// TIA Portal V20 export
// export: Created 2025-12-01T14:56:48.0251132Z, ExportSetting None, DisplayName Totally Integrated Automation Portal, DisplayVersion V20 Update 3, DisplayName TIA Portal Openness, DisplayVersion V20 Update 3, DisplayName TIA Portal Version Control Interface, DisplayVersion V20 Update 3, DisplayName STEP 7 Professional, DisplayVersion V20 Update 3, DisplayName STEP 7 Safety, DisplayVersion V20 Update 2, DisplayName WinCC Basic/Comfort/Advanced, DisplayVersion V20 Update 3, DisplayName WinCC Professional, DisplayVersion V20 Update 3, DisplayName WinCC Unified, DisplayVersion V20 Update 3
FUNCTION_BLOCK "FB101_GIRO_Mesa"   // FB101, LAD
TITLE = FB101
{ S7_Optimized_Access := 'FALSE' }
// FB complementaria a cualquier FB de mesa, solo gestiona el giro.
// stored: AutoNumber false, SetENOAutomatically false
   VAR_INPUT
      Mesa : UInt;   // Mesa de la FB
      Error_Tx : Bool;   // Error en el Tx
      EnTension : Bool;   // Existe Tension en la Mesa
      FalloVar_MG : Bool;   // Señal VAR ok
      MG_EnMovimiento : Bool;   // Señal VAR giro en curso
      PosMG_0 : Bool;   // Detector Posicion 0
      PosMG_90 : Bool;   // Detector Posicion 90
      PosMG_180 : Bool;   // Detector Posicion 180
      PosMG_270 : Bool;   // Detector Posicion 270
      pHsPR : Bool;   // pHs de Protrusion de la Mesa. Nota: No existe >> ON
      Movhabi0_90 : Bool;   // Habilitar zona movimiento entre 0 y 90º
      Movhabi90_180 : Bool;   // Habilitar zona movimiento entre 90 y 180º
      Movhabi180_270 : Bool;   // Habilitar zona movimiento entre 180 y 270º
      Movhabi270_0 : Bool;   // Habilitar zona movimiento entre 270 y 0º
      Mx_VelocidadLenta_In : Bool;   // Forzar velocidad lenta
      OrdPos_0 : Bool;   // Orden ir a Posicion 0
      OrdPos_90 : Bool;   // Orden ir a Posicion 90
      OrdPos_180 : Bool;   // Orden ir a Posicion 180
      OrdPos_270 : Bool;   // Orden ir a Posicion 270
      V_TOut_MG_90º : Int := 15;   // Timeout para un movimiento de 90º
      V_TOut_MG_180º : Int := 30;   // Timeout para un movimiento de 180º
      V_TOut_MG_270º : Int := 45;   // Timeout para un movimiento de 270º
      V_TOut_MG_BusqPos : Int := 15;   // Timeout para busqueda de posición en velo lenta
      V_CNT_PerdidaPos : Int := 5000;   // Perdida de posición
      V_PasoLenta_Mov90 : Int := 800;   // Cambio de velocidad durante un movimiento de 90º
      V_PasoLenta_Mov180 : Int := 1800;   // Cambio de velocidad durante un movimiento de 180º
      V_PasoLenta_Mov270 : Int := 2800;   // Cambio de velocidad durante un movimiento de 270º
      V_CNTSeg_AusPos : Int := 3000;   // Contador de seguridade posicionamiento
   END_VAR
   VAR
      MGiro_EnPos0 : Bool;   // Mesa Giro en posición 0º
      MGiro_EnPos90 : Bool;   // Mesa Giro en posición 90º
      MGiro_EnPos180 : Bool;   // Mesa Giro en posición 180º
      MGiro_EnPos270 : Bool;   // Mesa Giro en posición 270º
      PosOK { ExternalVisible := 'False'} : Bool;
      Orden_AvGiro : Bool;   // Orden de Avance (sentido agujas reloj)
      Orden_RtGiro : Bool;   // Orden de Retroceso (sentido inverso agujas reloj)
      DestinoPos0 : Bool;   // Destino a la posición 0º
      DestinoPos90 : Bool;   // Destino a la posición 90º
      DestinoPos180 : Bool;   // Destino a la posición 180º
      DestinoPos270 : Bool;   // Destino a la posición 270º
      Giro90º : Bool;   // Distancia de giro en grados desde origen hasta destino
      Giro180º : Bool;   // Distancia de giro en grados desde origen hasta destino
      Giro270º : Bool;   // Distancia de giro en grados desde origen hasta destino
      Pos_Desconocida : Bool;
      Pos_Conocida : Bool;
      Destino_Desconocido : Bool;
      Busq_Posicion : Bool;
      Mem_Busq_Posicion : Bool;
      VelocidadLenta { ExternalAccessible := 'False'; ExternalVisible := 'False'; ExternalWritable := 'False'} : Bool;
      MA_Avance_MG : Bool;   // Avance = ir de 0º a 360º
      MA_Retroceso_MG : Bool;   // Retroceso = volver de 360º a 0
      VelocidadRapida_MG : Bool;
      CNT_Paso_Lenta : Int;
      CNTSeg_AusPos { S7_SetPoint := 'True'} : "FB910_CNT_UHS";
      TMP_EnTension { S7_SetPoint := 'True'} : "FB910_CNT_UHS";
      TOut_MG { S7_SetPoint := 'True'} : "FB910_CNT_UHS";
      TOut_MG_BusPos { S7_SetPoint := 'True'} : "FB910_CNT_UHS";
      CNT_PerdidaPos { S7_SetPoint := 'True'} : "FB910_CNT_UHS";
   END_VAR
   VAR_TEMP
      EstadoZona : "EstadoZona";   // Estado de Zona de la Mesa
      EstadoVI : "EstadosMesa";   // Estado del Vehiculo Inteliguente de la Mesa
      ConfigFB : "UDT_ConfigFB";   // Configuracion de la FB de la Mesa
      V_TOut_MG : Int;
      Basura : Bool;
   END_VAR
   VAR_TEMP   // added for the SCL form of the ladder/FBD networks
      _w1 : Bool;
   END_VAR
BEGIN

REGION Network 1: INICIALIZAR - Recoger las Variables de Estado de la Mesa
   // Se recoge - Estado_CBx
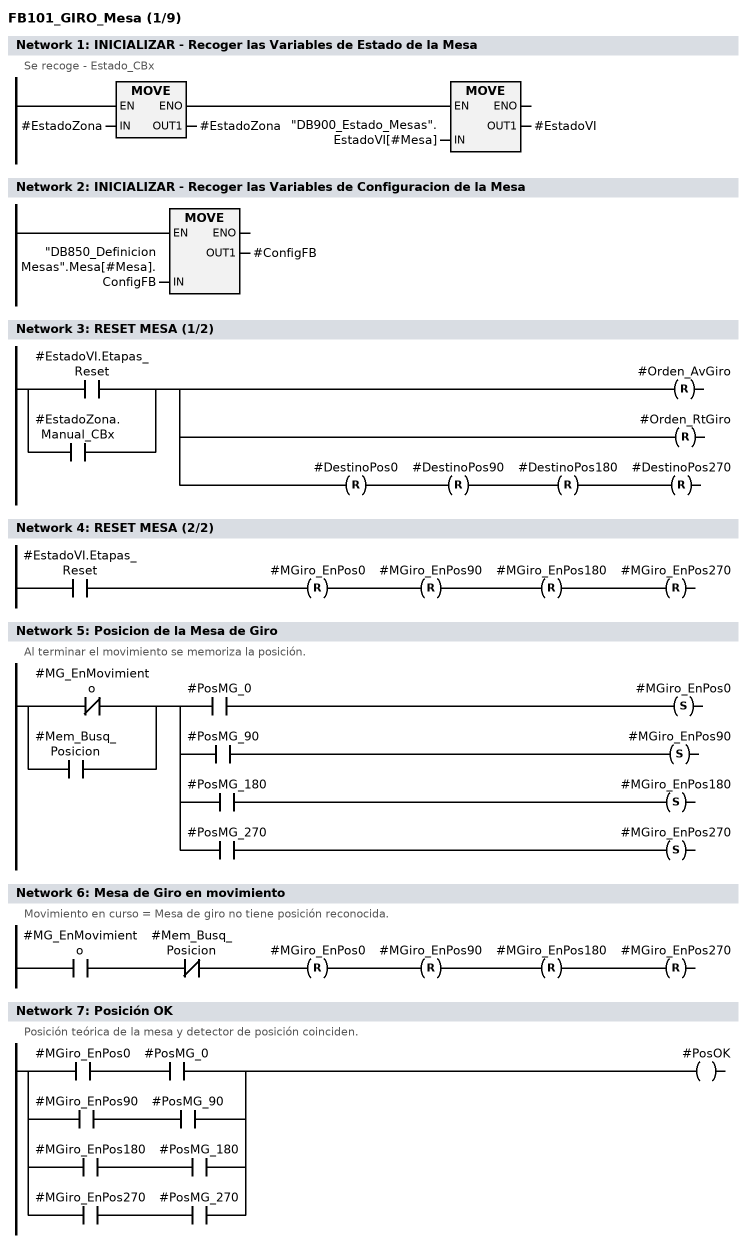
   RUNG wire#powerrail
      Move(in := #EstadoZona, out1 => #EstadoZona)
      Move(in := "DB900_Estado_Mesas".EstadoVI[#Mesa], out1 => #EstadoVI)
   END_RUNG
   // the same network as SCL:
   #EstadoZona := #EstadoZona;
   #EstadoVI := "DB900_Estado_Mesas".EstadoVI[#Mesa];
END_REGION

REGION Network 2: INICIALIZAR - Recoger las Variables de Configuracion de la Mesa
   RUNG wire#powerrail
      Move(in := "DB850_DefinicionMesas".Mesa[#Mesa].ConfigFB, out1 => #ConfigFB)
   END_RUNG
   // the same network as SCL:
   #ConfigFB := "DB850_DefinicionMesas".Mesa[#Mesa].ConfigFB;
END_REGION

REGION Network 3: RESET MESA (1/2)
   RUNG wire#powerrail
      Contact( #EstadoVI.Etapas_Reset )
      wire#w1
      R_Coil( #Orden_AvGiro )
   END_RUNG
   RUNG wire#powerrail
      Contact( #EstadoZona.Manual_CBx )
   END_RUNG wire#w1
   RUNG wire#w1
      R_Coil( #Orden_RtGiro )
   END_RUNG
   RUNG wire#w1
      R_Coil( #DestinoPos0 )
      R_Coil( #DestinoPos90 )
      R_Coil( #DestinoPos180 )
      R_Coil( #DestinoPos270 )
   END_RUNG
   // the same network as SCL:
   IF #EstadoVI.Etapas_Reset OR #EstadoZona.Manual_CBx THEN
       #Orden_AvGiro := FALSE;
       #Orden_RtGiro := FALSE;
       #DestinoPos0 := FALSE;
       #DestinoPos90 := FALSE;
       #DestinoPos180 := FALSE;
       #DestinoPos270 := FALSE;
   END_IF;
END_REGION

REGION Network 4: RESET MESA (2/2)
   RUNG wire#powerrail
      Contact( #EstadoVI.Etapas_Reset )
      R_Coil( #MGiro_EnPos0 )
      R_Coil( #MGiro_EnPos90 )
      R_Coil( #MGiro_EnPos180 )
      R_Coil( #MGiro_EnPos270 )
   END_RUNG
   // the same network as SCL:
   IF #EstadoVI.Etapas_Reset THEN
       #MGiro_EnPos0 := FALSE;
       #MGiro_EnPos90 := FALSE;
       #MGiro_EnPos180 := FALSE;
       #MGiro_EnPos270 := FALSE;
   END_IF;
END_REGION

REGION Network 5: Posicion de la Mesa de Giro
   // Al terminar el movimiento se memoriza la posición.
   RUNG wire#powerrail
      I_Contact( #MG_EnMovimiento )
      wire#w1
      Contact( #PosMG_0 )
      S_Coil( #MGiro_EnPos0 )
   END_RUNG
   RUNG wire#powerrail
      Contact( #Mem_Busq_Posicion )
   END_RUNG wire#w1
   RUNG wire#w1
      Contact( #PosMG_90 )
      S_Coil( #MGiro_EnPos90 )
   END_RUNG
   RUNG wire#w1
      Contact( #PosMG_180 )
      S_Coil( #MGiro_EnPos180 )
   END_RUNG
   RUNG wire#w1
      Contact( #PosMG_270 )
      S_Coil( #MGiro_EnPos270 )
   END_RUNG
   // the same network as SCL:
   #_w1 := NOT #MG_EnMovimiento OR #Mem_Busq_Posicion;
   IF #_w1 AND #PosMG_0 THEN #MGiro_EnPos0 := TRUE; END_IF;
   IF #_w1 AND #PosMG_90 THEN #MGiro_EnPos90 := TRUE; END_IF;
   IF #_w1 AND #PosMG_180 THEN #MGiro_EnPos180 := TRUE; END_IF;
   IF #_w1 AND #PosMG_270 THEN #MGiro_EnPos270 := TRUE; END_IF;
END_REGION

REGION Network 6: Mesa de Giro en movimiento
   // Movimiento en curso = Mesa de giro no tiene posición reconocida.
   RUNG wire#powerrail
      Contact( #MG_EnMovimiento )
      I_Contact( #Mem_Busq_Posicion )
      R_Coil( #MGiro_EnPos0 )
      R_Coil( #MGiro_EnPos90 )
      R_Coil( #MGiro_EnPos180 )
      R_Coil( #MGiro_EnPos270 )
   END_RUNG
   // the same network as SCL:
   IF #MG_EnMovimiento AND NOT #Mem_Busq_Posicion THEN
       #MGiro_EnPos0 := FALSE;
       #MGiro_EnPos90 := FALSE;
       #MGiro_EnPos180 := FALSE;
       #MGiro_EnPos270 := FALSE;
   END_IF;
END_REGION

REGION Network 7: Posición OK
   // Posición teórica de la mesa y detector de posición coinciden.
   RUNG wire#powerrail
      Contact( #MGiro_EnPos0 )
      Contact( #PosMG_0 )
      wire#w1
      Coil( #PosOK )
   END_RUNG
   RUNG wire#powerrail
      Contact( #MGiro_EnPos90 )
      Contact( #PosMG_90 )
   END_RUNG wire#w1
   RUNG wire#powerrail
      Contact( #MGiro_EnPos180 )
      Contact( #PosMG_180 )
   END_RUNG wire#w1
   RUNG wire#powerrail
      Contact( #MGiro_EnPos270 )
      Contact( #PosMG_270 )
   END_RUNG wire#w1
   // the same network as SCL:
   #PosOK := (#MGiro_EnPos0 AND #PosMG_0) OR (#MGiro_EnPos90 AND #PosMG_90) OR (#MGiro_EnPos180 AND #PosMG_180) OR (#MGiro_EnPos270 AND #PosMG_270);
END_REGION

REGION Network 8: Destino Desconocido // Posicion desconocida // Posicion Conocida
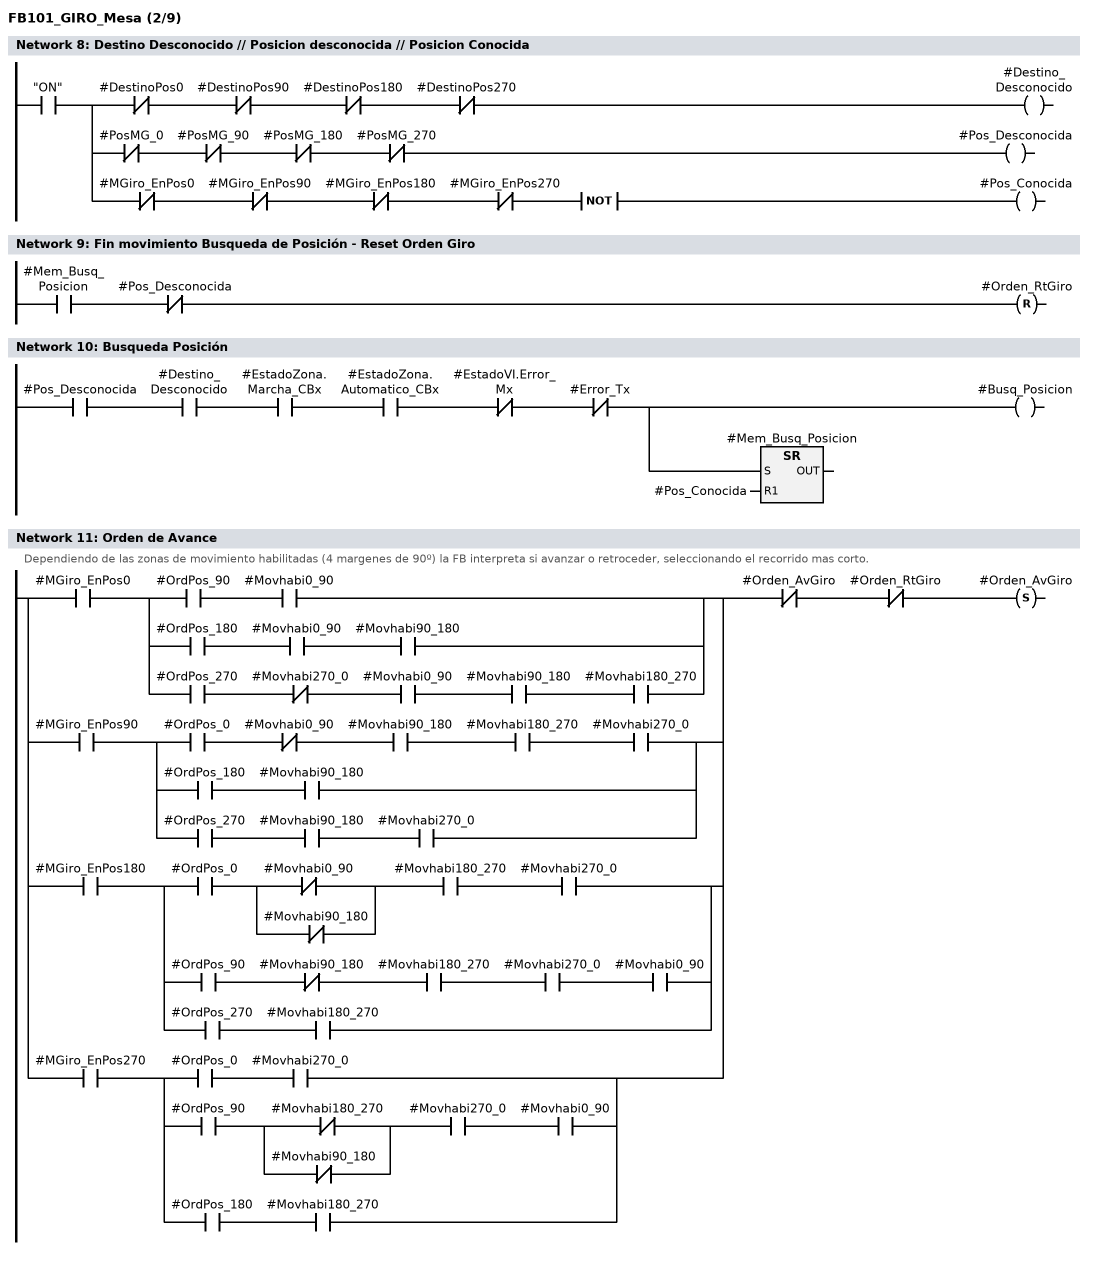
   RUNG wire#powerrail
      Contact( "ON" )
      wire#w1
      I_Contact( #DestinoPos0 )
      I_Contact( #DestinoPos90 )
      I_Contact( #DestinoPos180 )
      I_Contact( #DestinoPos270 )
      Coil( #Destino_Desconocido )
   END_RUNG
   RUNG wire#w1
      I_Contact( #PosMG_0 )
      I_Contact( #PosMG_90 )
      I_Contact( #PosMG_180 )
      I_Contact( #PosMG_270 )
      Coil( #Pos_Desconocida )
   END_RUNG
   RUNG wire#w1
      I_Contact( #MGiro_EnPos0 )
      I_Contact( #MGiro_EnPos90 )
      I_Contact( #MGiro_EnPos180 )
      I_Contact( #MGiro_EnPos270 )
      Not()
      Coil( #Pos_Conocida )
   END_RUNG
   // the same network as SCL:
   #Destino_Desconocido := "ON" AND NOT #DestinoPos0 AND NOT #DestinoPos90 AND NOT #DestinoPos180 AND NOT #DestinoPos270;
   #Pos_Desconocida := "ON" AND NOT #PosMG_0 AND NOT #PosMG_90 AND NOT #PosMG_180 AND NOT #PosMG_270;
   #Pos_Conocida := NOT ("ON" AND NOT #MGiro_EnPos0 AND NOT #MGiro_EnPos90 AND NOT #MGiro_EnPos180 AND NOT #MGiro_EnPos270);
END_REGION

REGION Network 9: Fin movimiento Busqueda de Posición - Reset Orden Giro
   RUNG wire#powerrail
      Contact( #Mem_Busq_Posicion )
      I_Contact( #Pos_Desconocida )
      R_Coil( #Orden_RtGiro )
   END_RUNG
   // the same network as SCL:
   IF #Mem_Busq_Posicion AND NOT #Pos_Desconocida THEN #Orden_RtGiro := FALSE; END_IF;
END_REGION

REGION Network 10: Busqueda Posición
   RUNG wire#powerrail
      Contact( #Pos_Desconocida )
      Contact( #Destino_Desconocido )
      Contact( #EstadoZona.Marcha_CBx )
      Contact( #EstadoZona.Automatico_CBx )
      I_Contact( #EstadoVI.Error_Mx )
      I_Contact( #Error_Tx )
      wire#w1
      Coil( #Busq_Posicion )
   END_RUNG
   RUNG wire#w1
      S_SR(operand := #Mem_Busq_Posicion, r1 := #Pos_Conocida)
   END_RUNG
   // the same network as SCL:
   #Busq_Posicion := #Pos_Desconocida AND #Destino_Desconocido AND #EstadoZona.Marcha_CBx AND #EstadoZona.Automatico_CBx AND NOT #EstadoVI.Error_Mx AND NOT #Error_Tx;
   IF #Busq_Posicion THEN
       #Mem_Busq_Posicion := TRUE;   // SR flip-flop
   END_IF;
   IF #Pos_Conocida THEN #Mem_Busq_Posicion := FALSE; END_IF;
END_REGION

REGION Network 11: Orden de Avance
   // Dependiendo de las zonas de movimiento habilitadas (4 margenes de 90º) la FB interpreta si avanzar o retroceder, seleccionando el recorrido mas corto.
   RUNG wire#powerrail
      Contact( #MGiro_EnPos0 )
      wire#w1
      Contact( #OrdPos_90 )
      Contact( #Movhabi0_90 )
      wire#w2
      I_Contact( #Orden_AvGiro )
      I_Contact( #Orden_RtGiro )
      S_Coil( #Orden_AvGiro )
   END_RUNG
   RUNG wire#w1
      Contact( #OrdPos_180 )
      Contact( #Movhabi0_90 )
      Contact( #Movhabi90_180 )
   END_RUNG wire#w2
   RUNG wire#w1
      Contact( #OrdPos_270 )
      I_Contact( #Movhabi270_0 )
      Contact( #Movhabi0_90 )
      Contact( #Movhabi90_180 )
      Contact( #Movhabi180_270 )
   END_RUNG wire#w2
   RUNG wire#powerrail
      Contact( #MGiro_EnPos90 )
      wire#w3
      Contact( #OrdPos_0 )
      I_Contact( #Movhabi0_90 )
      Contact( #Movhabi90_180 )
      Contact( #Movhabi180_270 )
      Contact( #Movhabi270_0 )
   END_RUNG wire#w2
   RUNG wire#w3
      Contact( #OrdPos_180 )
      Contact( #Movhabi90_180 )
   END_RUNG wire#w2
   RUNG wire#w3
      Contact( #OrdPos_270 )
      Contact( #Movhabi90_180 )
      Contact( #Movhabi270_0 )
   END_RUNG wire#w2
   RUNG wire#powerrail
      Contact( #MGiro_EnPos180 )
      wire#w4
      Contact( #OrdPos_0 )
      wire#w5
      I_Contact( #Movhabi0_90 )
      wire#w6
      Contact( #Movhabi180_270 )
      Contact( #Movhabi270_0 )
   END_RUNG wire#w2
   RUNG wire#w5
      I_Contact( #Movhabi90_180 )
   END_RUNG wire#w6
   RUNG wire#w4
      Contact( #OrdPos_90 )
      I_Contact( #Movhabi90_180 )
      Contact( #Movhabi180_270 )
      Contact( #Movhabi270_0 )
      Contact( #Movhabi0_90 )
   END_RUNG wire#w2
   RUNG wire#w4
      Contact( #OrdPos_270 )
      Contact( #Movhabi180_270 )
   END_RUNG wire#w2
   RUNG wire#powerrail
      Contact( #MGiro_EnPos270 )
      wire#w7
      Contact( #OrdPos_0 )
      Contact( #Movhabi270_0 )
   END_RUNG wire#w2
   RUNG wire#w7
      Contact( #OrdPos_90 )
      wire#w8
      I_Contact( #Movhabi180_270 )
      wire#w9
      Contact( #Movhabi270_0 )
      Contact( #Movhabi0_90 )
   END_RUNG wire#w2
   RUNG wire#w8
      I_Contact( #Movhabi90_180 )
   END_RUNG wire#w9
   RUNG wire#w7
      Contact( #OrdPos_180 )
      Contact( #Movhabi180_270 )
   END_RUNG wire#w2
   // the same network as SCL:
   IF ((#MGiro_EnPos0 AND ((#OrdPos_90 AND #Movhabi0_90) OR (#OrdPos_180 AND #Movhabi0_90 AND #Movhabi90_180) OR (#OrdPos_270 AND NOT #Movhabi270_0 AND #Movhabi0_90 AND #Movhabi90_180 AND #Movhabi180_270))) OR (#MGiro_EnPos90 AND ((#OrdPos_0 AND NOT #Movhabi0_90 AND #Movhabi90_180 AND #Movhabi180_270 AND #Movhabi270_0) OR (#OrdPos_180 AND #Movhabi90_180) OR (#OrdPos_270 AND #Movhabi90_180 AND #Movhabi270_0))) OR (#MGiro_EnPos180 AND ((#OrdPos_0 AND (NOT #Movhabi0_90 OR NOT #Movhabi90_180) AND #Movhabi180_270 AND #Movhabi270_0) OR (#OrdPos_90 AND NOT #Movhabi90_180 AND #Movhabi180_270 AND #Movhabi270_0 AND #Movhabi0_90) OR (#OrdPos_270 AND #Movhabi180_270))) OR (#MGiro_EnPos270 AND ((#OrdPos_0 AND #Movhabi270_0) OR (#OrdPos_90 AND (NOT #Movhabi180_270 OR NOT #Movhabi90_180) AND #Movhabi270_0 AND #Movhabi0_90) OR (#OrdPos_180 AND #Movhabi180_270)))) AND NOT #Orden_AvGiro AND NOT #Orden_RtGiro THEN
       #Orden_AvGiro := TRUE;
   END_IF;
END_REGION

REGION Network 12: Orden de Retroceso
   // Dependiendo de las zonas de movimiento habilitadas (4 margenes de 90º) la FB interpreta si avanzar o retroceder, seleccionando el recorrido mas corto.
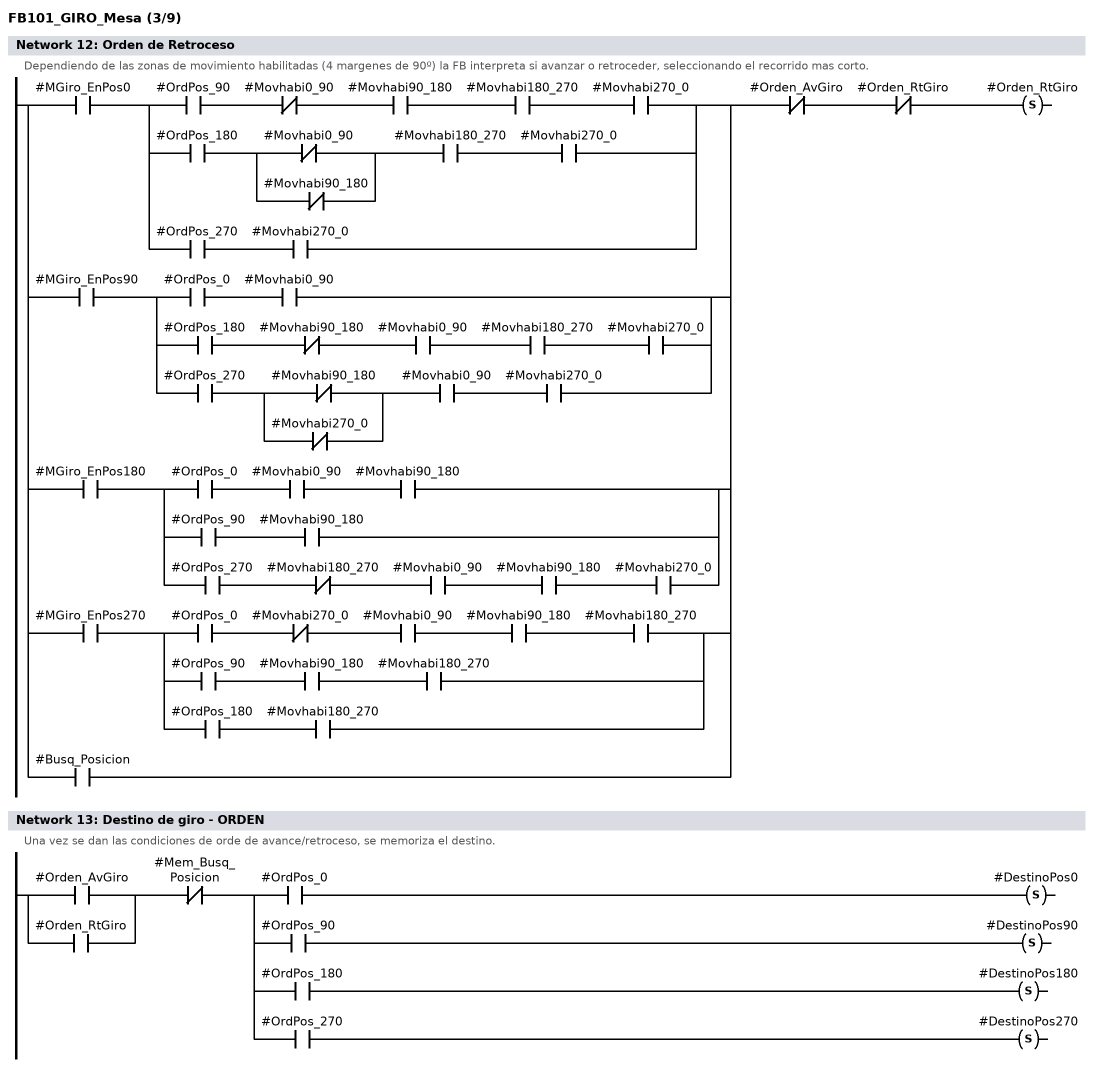
   RUNG wire#powerrail
      Contact( #MGiro_EnPos0 )
      wire#w1
      Contact( #OrdPos_90 )
      I_Contact( #Movhabi0_90 )
      Contact( #Movhabi90_180 )
      Contact( #Movhabi180_270 )
      Contact( #Movhabi270_0 )
      wire#w2
      I_Contact( #Orden_AvGiro )
      I_Contact( #Orden_RtGiro )
      S_Coil( #Orden_RtGiro )
   END_RUNG
   RUNG wire#w1
      Contact( #OrdPos_180 )
      wire#w3
      I_Contact( #Movhabi0_90 )
      wire#w4
      Contact( #Movhabi180_270 )
      Contact( #Movhabi270_0 )
   END_RUNG wire#w2
   RUNG wire#w3
      I_Contact( #Movhabi90_180 )
   END_RUNG wire#w4
   RUNG wire#w1
      Contact( #OrdPos_270 )
      Contact( #Movhabi270_0 )
   END_RUNG wire#w2
   RUNG wire#powerrail
      Contact( #MGiro_EnPos90 )
      wire#w5
      Contact( #OrdPos_0 )
      Contact( #Movhabi0_90 )
   END_RUNG wire#w2
   RUNG wire#w5
      Contact( #OrdPos_180 )
      I_Contact( #Movhabi90_180 )
      Contact( #Movhabi0_90 )
      Contact( #Movhabi180_270 )
      Contact( #Movhabi270_0 )
   END_RUNG wire#w2
   RUNG wire#w5
      Contact( #OrdPos_270 )
      wire#w6
      I_Contact( #Movhabi90_180 )
      wire#w7
      Contact( #Movhabi0_90 )
      Contact( #Movhabi270_0 )
   END_RUNG wire#w2
   RUNG wire#w6
      I_Contact( #Movhabi270_0 )
   END_RUNG wire#w7
   RUNG wire#powerrail
      Contact( #MGiro_EnPos180 )
      wire#w8
      Contact( #OrdPos_0 )
      Contact( #Movhabi0_90 )
      Contact( #Movhabi90_180 )
   END_RUNG wire#w2
   RUNG wire#w8
      Contact( #OrdPos_90 )
      Contact( #Movhabi90_180 )
   END_RUNG wire#w2
   RUNG wire#w8
      Contact( #OrdPos_270 )
      I_Contact( #Movhabi180_270 )
      Contact( #Movhabi0_90 )
      Contact( #Movhabi90_180 )
      Contact( #Movhabi270_0 )
   END_RUNG wire#w2
   RUNG wire#powerrail
      Contact( #MGiro_EnPos270 )
      wire#w9
      Contact( #OrdPos_0 )
      I_Contact( #Movhabi270_0 )
      Contact( #Movhabi0_90 )
      Contact( #Movhabi90_180 )
      Contact( #Movhabi180_270 )
   END_RUNG wire#w2
   RUNG wire#w9
      Contact( #OrdPos_90 )
      Contact( #Movhabi90_180 )
      Contact( #Movhabi180_270 )
   END_RUNG wire#w2
   RUNG wire#w9
      Contact( #OrdPos_180 )
      Contact( #Movhabi180_270 )
   END_RUNG wire#w2
   RUNG wire#powerrail
      Contact( #Busq_Posicion )
   END_RUNG wire#w2
   // the same network as SCL:
   IF ((#MGiro_EnPos0 AND ((#OrdPos_90 AND NOT #Movhabi0_90 AND #Movhabi90_180 AND #Movhabi180_270 AND #Movhabi270_0) OR (#OrdPos_180 AND (NOT #Movhabi0_90 OR NOT #Movhabi90_180) AND #Movhabi180_270 AND #Movhabi270_0) OR (#OrdPos_270 AND #Movhabi270_0))) OR (#MGiro_EnPos90 AND ((#OrdPos_0 AND #Movhabi0_90) OR (#OrdPos_180 AND NOT #Movhabi90_180 AND #Movhabi0_90 AND #Movhabi180_270 AND #Movhabi270_0) OR (#OrdPos_270 AND (NOT #Movhabi90_180 OR NOT #Movhabi270_0) AND #Movhabi0_90 AND #Movhabi270_0))) OR (#MGiro_EnPos180 AND ((#OrdPos_0 AND #Movhabi0_90 AND #Movhabi90_180) OR (#OrdPos_90 AND #Movhabi90_180) OR (#OrdPos_270 AND NOT #Movhabi180_270 AND #Movhabi0_90 AND #Movhabi90_180 AND #Movhabi270_0))) OR (#MGiro_EnPos270 AND ((#OrdPos_0 AND NOT #Movhabi270_0 AND #Movhabi0_90 AND #Movhabi90_180 AND #Movhabi180_270) OR (#OrdPos_90 AND #Movhabi90_180 AND #Movhabi180_270) OR (#OrdPos_180 AND #Movhabi180_270))) OR #Busq_Posicion) AND NOT #Orden_AvGiro AND NOT #Orden_RtGiro THEN
       #Orden_RtGiro := TRUE;
   END_IF;
END_REGION

REGION Network 13: Destino de giro - ORDEN
   // Una vez se dan las condiciones de orde de avance/retroceso, se memoriza el destino.
   RUNG wire#powerrail
      Contact( #Orden_AvGiro )
      wire#w1
      I_Contact( #Mem_Busq_Posicion )
      wire#w2
      Contact( #OrdPos_0 )
      S_Coil( #DestinoPos0 )
   END_RUNG
   RUNG wire#powerrail
      Contact( #Orden_RtGiro )
   END_RUNG wire#w1
   RUNG wire#w2
      Contact( #OrdPos_90 )
      S_Coil( #DestinoPos90 )
   END_RUNG
   RUNG wire#w2
      Contact( #OrdPos_180 )
      S_Coil( #DestinoPos180 )
   END_RUNG
   RUNG wire#w2
      Contact( #OrdPos_270 )
      S_Coil( #DestinoPos270 )
   END_RUNG
   // the same network as SCL:
   #_w1 := (#Orden_AvGiro OR #Orden_RtGiro) AND NOT #Mem_Busq_Posicion;
   IF #_w1 AND #OrdPos_0 THEN #DestinoPos0 := TRUE; END_IF;
   IF #_w1 AND #OrdPos_90 THEN #DestinoPos90 := TRUE; END_IF;
   IF #_w1 AND #OrdPos_180 THEN #DestinoPos180 := TRUE; END_IF;
   IF #_w1 AND #OrdPos_270 THEN #DestinoPos270 := TRUE; END_IF;
END_REGION

REGION Network 14: Destino de giro - FIN
   // Al llegar a posición el destino se borra.
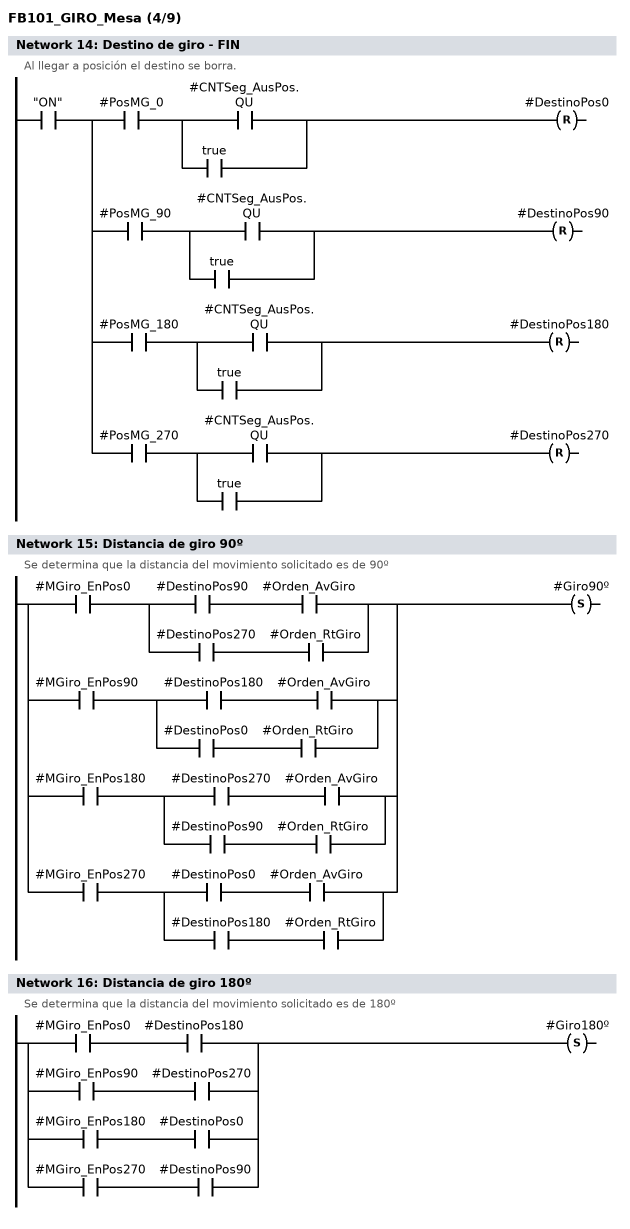
   RUNG wire#powerrail
      Contact( "ON" )
      wire#w1
      Contact( #PosMG_0 )
      wire#w2
      Contact( #CNTSeg_AusPos.QU )
      wire#w3
      R_Coil( #DestinoPos0 )
   END_RUNG
   RUNG wire#w2
      Contact( true )
   END_RUNG wire#w3
   RUNG wire#w1
      Contact( #PosMG_90 )
      wire#w4
      Contact( #CNTSeg_AusPos.QU )
      wire#w5
      R_Coil( #DestinoPos90 )
   END_RUNG
   RUNG wire#w4
      Contact( true )
   END_RUNG wire#w5
   RUNG wire#w1
      Contact( #PosMG_180 )
      wire#w6
      Contact( #CNTSeg_AusPos.QU )
      wire#w7
      R_Coil( #DestinoPos180 )
   END_RUNG
   RUNG wire#w6
      Contact( true )
   END_RUNG wire#w7
   RUNG wire#w1
      Contact( #PosMG_270 )
      wire#w8
      Contact( #CNTSeg_AusPos.QU )
      wire#w9
      R_Coil( #DestinoPos270 )
   END_RUNG
   RUNG wire#w8
      Contact( true )
   END_RUNG wire#w9
   // the same network as SCL:
   IF "ON" AND #PosMG_0 AND (#CNTSeg_AusPos.QU OR true) THEN #DestinoPos0 := FALSE; END_IF;
   IF "ON" AND #PosMG_90 AND (#CNTSeg_AusPos.QU OR true) THEN #DestinoPos90 := FALSE; END_IF;
   IF "ON" AND #PosMG_180 AND (#CNTSeg_AusPos.QU OR true) THEN #DestinoPos180 := FALSE; END_IF;
   IF "ON" AND #PosMG_270 AND (#CNTSeg_AusPos.QU OR true) THEN #DestinoPos270 := FALSE; END_IF;
END_REGION

REGION Network 15: Distancia de giro 90º
   // Se determina que la distancia del movimiento solicitado es de 90º
   RUNG wire#powerrail
      Contact( #MGiro_EnPos0 )
      wire#w1
      Contact( #DestinoPos90 )
      Contact( #Orden_AvGiro )
      wire#w2
      S_Coil( #Giro90º )
   END_RUNG
   RUNG wire#w1
      Contact( #DestinoPos270 )
      Contact( #Orden_RtGiro )
   END_RUNG wire#w2
   RUNG wire#powerrail
      Contact( #MGiro_EnPos90 )
      wire#w3
      Contact( #DestinoPos180 )
      Contact( #Orden_AvGiro )
   END_RUNG wire#w2
   RUNG wire#w3
      Contact( #DestinoPos0 )
      Contact( #Orden_RtGiro )
   END_RUNG wire#w2
   RUNG wire#powerrail
      Contact( #MGiro_EnPos180 )
      wire#w4
      Contact( #DestinoPos270 )
      Contact( #Orden_AvGiro )
   END_RUNG wire#w2
   RUNG wire#w4
      Contact( #DestinoPos90 )
      Contact( #Orden_RtGiro )
   END_RUNG wire#w2
   RUNG wire#powerrail
      Contact( #MGiro_EnPos270 )
      wire#w5
      Contact( #DestinoPos0 )
      Contact( #Orden_AvGiro )
   END_RUNG wire#w2
   RUNG wire#w5
      Contact( #DestinoPos180 )
      Contact( #Orden_RtGiro )
   END_RUNG wire#w2
   // the same network as SCL:
   IF (#MGiro_EnPos0 AND ((#DestinoPos90 AND #Orden_AvGiro) OR (#DestinoPos270 AND #Orden_RtGiro))) OR (#MGiro_EnPos90 AND ((#DestinoPos180 AND #Orden_AvGiro) OR (#DestinoPos0 AND #Orden_RtGiro))) OR (#MGiro_EnPos180 AND ((#DestinoPos270 AND #Orden_AvGiro) OR (#DestinoPos90 AND #Orden_RtGiro))) OR (#MGiro_EnPos270 AND ((#DestinoPos0 AND #Orden_AvGiro) OR (#DestinoPos180 AND #Orden_RtGiro))) THEN
       #Giro90º := TRUE;
   END_IF;
END_REGION

REGION Network 16: Distancia de giro 180º
   // Se determina que la distancia del movimiento solicitado es de 180º
   RUNG wire#powerrail
      Contact( #MGiro_EnPos0 )
      Contact( #DestinoPos180 )
      wire#w1
      S_Coil( #Giro180º )
   END_RUNG
   RUNG wire#powerrail
      Contact( #MGiro_EnPos90 )
      Contact( #DestinoPos270 )
   END_RUNG wire#w1
   RUNG wire#powerrail
      Contact( #MGiro_EnPos180 )
      Contact( #DestinoPos0 )
   END_RUNG wire#w1
   RUNG wire#powerrail
      Contact( #MGiro_EnPos270 )
      Contact( #DestinoPos90 )
   END_RUNG wire#w1
   // the same network as SCL:
   IF (#MGiro_EnPos0 AND #DestinoPos180) OR (#MGiro_EnPos90 AND #DestinoPos270) OR (#MGiro_EnPos180 AND #DestinoPos0) OR (#MGiro_EnPos270 AND #DestinoPos90) THEN
       #Giro180º := TRUE;
   END_IF;
END_REGION

REGION Network 17: Distancia de giro 270º
   // Se determina que la distancia del movimiento solicitado es de 270º
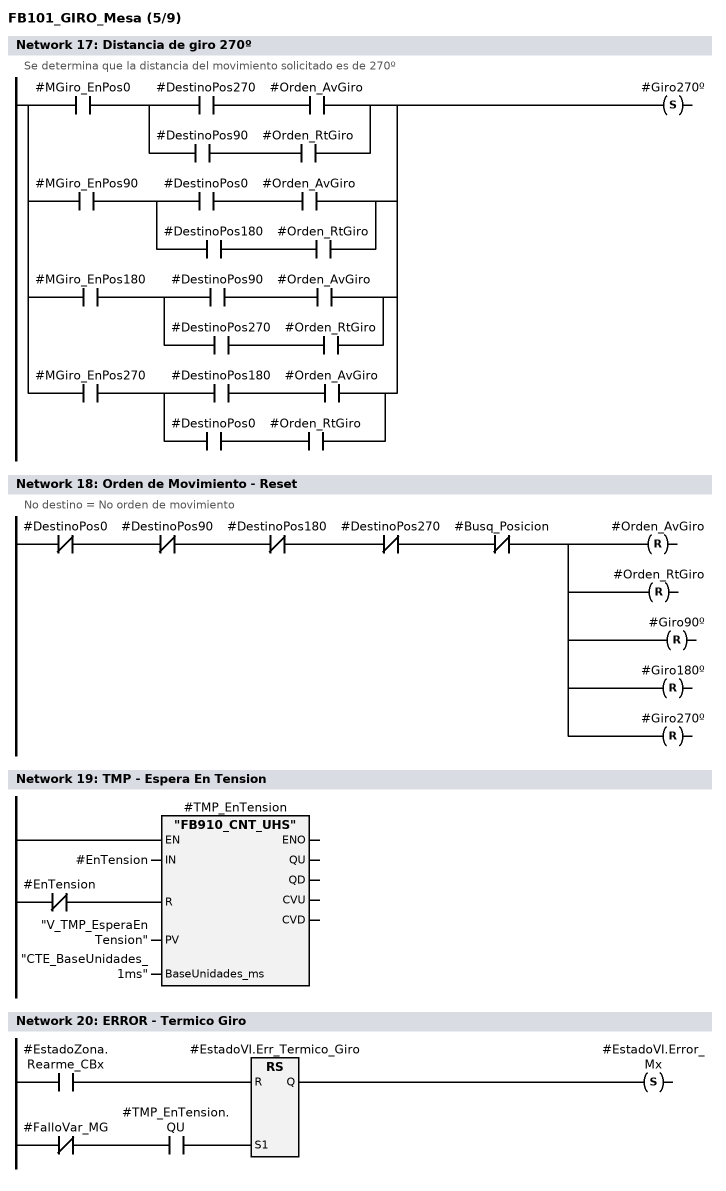
   RUNG wire#powerrail
      Contact( #MGiro_EnPos0 )
      wire#w1
      Contact( #DestinoPos270 )
      Contact( #Orden_AvGiro )
      wire#w2
      S_Coil( #Giro270º )
   END_RUNG
   RUNG wire#w1
      Contact( #DestinoPos90 )
      Contact( #Orden_RtGiro )
   END_RUNG wire#w2
   RUNG wire#powerrail
      Contact( #MGiro_EnPos90 )
      wire#w3
      Contact( #DestinoPos0 )
      Contact( #Orden_AvGiro )
   END_RUNG wire#w2
   RUNG wire#w3
      Contact( #DestinoPos180 )
      Contact( #Orden_RtGiro )
   END_RUNG wire#w2
   RUNG wire#powerrail
      Contact( #MGiro_EnPos180 )
      wire#w4
      Contact( #DestinoPos90 )
      Contact( #Orden_AvGiro )
   END_RUNG wire#w2
   RUNG wire#w4
      Contact( #DestinoPos270 )
      Contact( #Orden_RtGiro )
   END_RUNG wire#w2
   RUNG wire#powerrail
      Contact( #MGiro_EnPos270 )
      wire#w5
      Contact( #DestinoPos180 )
      Contact( #Orden_AvGiro )
   END_RUNG wire#w2
   RUNG wire#w5
      Contact( #DestinoPos0 )
      Contact( #Orden_RtGiro )
   END_RUNG wire#w2
   // the same network as SCL:
   IF (#MGiro_EnPos0 AND ((#DestinoPos270 AND #Orden_AvGiro) OR (#DestinoPos90 AND #Orden_RtGiro))) OR (#MGiro_EnPos90 AND ((#DestinoPos0 AND #Orden_AvGiro) OR (#DestinoPos180 AND #Orden_RtGiro))) OR (#MGiro_EnPos180 AND ((#DestinoPos90 AND #Orden_AvGiro) OR (#DestinoPos270 AND #Orden_RtGiro))) OR (#MGiro_EnPos270 AND ((#DestinoPos180 AND #Orden_AvGiro) OR (#DestinoPos0 AND #Orden_RtGiro))) THEN
       #Giro270º := TRUE;
   END_IF;
END_REGION

REGION Network 18: Orden de Movimiento - Reset
   // No destino = No orden de movimiento
   RUNG wire#powerrail
      I_Contact( #DestinoPos0 )
      I_Contact( #DestinoPos90 )
      I_Contact( #DestinoPos180 )
      I_Contact( #DestinoPos270 )
      I_Contact( #Busq_Posicion )
      wire#w1
      R_Coil( #Orden_AvGiro )
   END_RUNG
   RUNG wire#w1
      R_Coil( #Orden_RtGiro )
   END_RUNG
   RUNG wire#w1
      R_Coil( #Giro90º )
   END_RUNG
   RUNG wire#w1
      R_Coil( #Giro180º )
   END_RUNG
   RUNG wire#w1
      R_Coil( #Giro270º )
   END_RUNG
   // the same network as SCL:
   IF NOT #DestinoPos0 AND NOT #DestinoPos90 AND NOT #DestinoPos180 AND NOT #DestinoPos270 AND NOT #Busq_Posicion THEN
       #Orden_AvGiro := FALSE;
       #Orden_RtGiro := FALSE;
       #Giro90º := FALSE;
       #Giro180º := FALSE;
       #Giro270º := FALSE;
   END_IF;
END_REGION

REGION Network 19: TMP - Espera En Tension
   RUNG wire#powerrail
      #TMP_EnTension(R := wire#w1, IN := #EnTension, PV := "V_TMP_EsperaEnTension", BaseUnidades_ms := "CTE_BaseUnidades_1ms", QU =>, QD =>, CVU =>, CVD =>)
   END_RUNG
   RUNG wire#powerrail
      I_Contact( #EnTension )
   END_RUNG wire#w1
   // the same network as SCL:
   #TMP_EnTension(IN := #EnTension,   // "FB910_CNT_UHS"
                  R := NOT #EnTension,
                  PV := "V_TMP_EsperaEnTension",
                  BaseUnidades_ms := "CTE_BaseUnidades_1ms");
END_REGION

REGION Network 20: ERROR - Termico Giro
   RUNG wire#powerrail
      Contact( #EstadoZona.Rearme_CBx )
      S_RS(operand := #EstadoVI.Err_Termico_Giro, s1 := wire#w1)
      S_Coil( #EstadoVI.Error_Mx )
   END_RUNG
   RUNG wire#powerrail
      I_Contact( #FalloVar_MG )
      Contact( #TMP_EnTension.QU )
   END_RUNG wire#w1
   // the same network as SCL:
   IF #EstadoZona.Rearme_CBx THEN
       #EstadoVI.Err_Termico_Giro := FALSE;   // RS flip-flop
   END_IF;
   IF NOT #FalloVar_MG AND #TMP_EnTension.QU THEN #EstadoVI.Err_Termico_Giro := TRUE; END_IF;
   IF #EstadoVI.Err_Termico_Giro THEN #EstadoVI.Error_Mx := TRUE; END_IF;
END_REGION

REGION Network 21: ERROR - Protusion
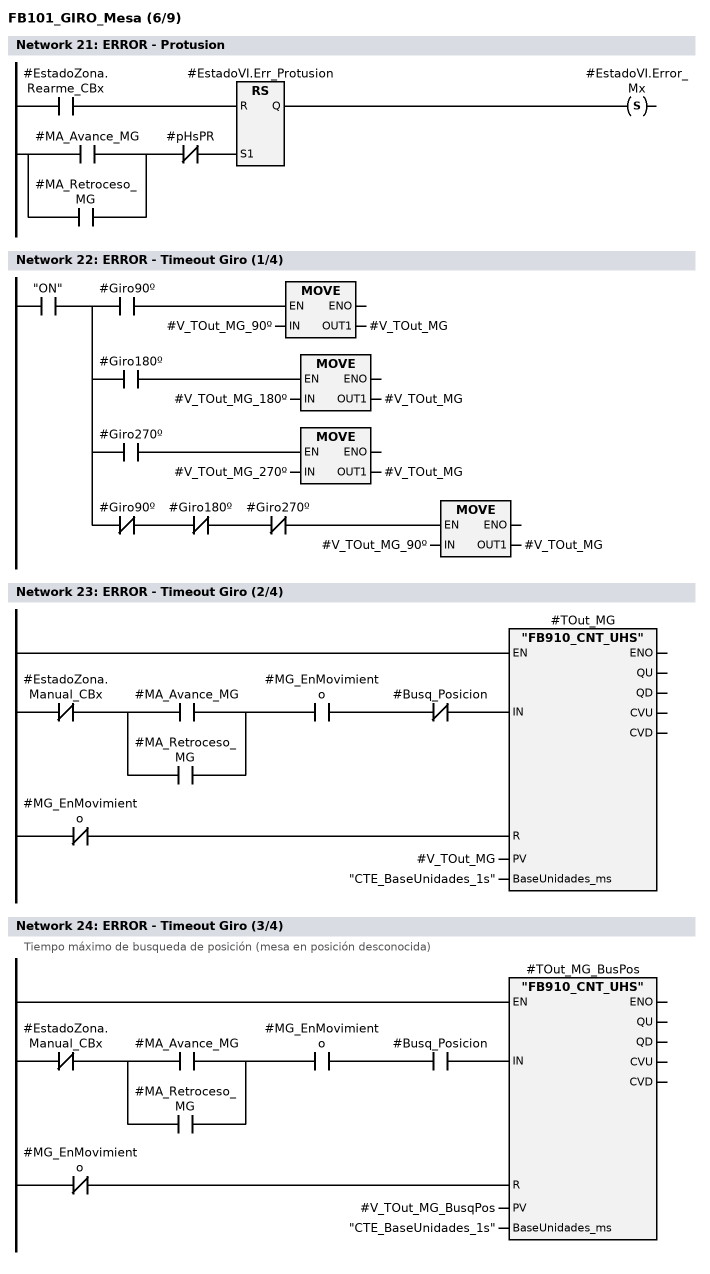
   RUNG wire#powerrail
      Contact( #EstadoZona.Rearme_CBx )
      S_RS(operand := #EstadoVI.Err_Protusion, s1 := wire#w2)
      S_Coil( #EstadoVI.Error_Mx )
   END_RUNG
   RUNG wire#powerrail
      Contact( #MA_Avance_MG )
      wire#w1
      I_Contact( #pHsPR )
   END_RUNG wire#w2
   RUNG wire#powerrail
      Contact( #MA_Retroceso_MG )
   END_RUNG wire#w1
   // the same network as SCL:
   IF #EstadoZona.Rearme_CBx THEN
       #EstadoVI.Err_Protusion := FALSE;   // RS flip-flop
   END_IF;
   IF (#MA_Avance_MG OR #MA_Retroceso_MG) AND NOT #pHsPR THEN #EstadoVI.Err_Protusion := TRUE; END_IF;
   IF #EstadoVI.Err_Protusion THEN #EstadoVI.Error_Mx := TRUE; END_IF;
END_REGION

REGION Network 22: ERROR - Timeout Giro (1/4)
   RUNG wire#powerrail
      Contact( "ON" )
      wire#w1
      Contact( #Giro90º )
      Move(in := #V_TOut_MG_90º, out1 => #V_TOut_MG)
   END_RUNG
   RUNG wire#w1
      Contact( #Giro180º )
      Move(in := #V_TOut_MG_180º, out1 => #V_TOut_MG)
   END_RUNG
   RUNG wire#w1
      Contact( #Giro270º )
      Move(in := #V_TOut_MG_270º, out1 => #V_TOut_MG)
   END_RUNG
   RUNG wire#w1
      I_Contact( #Giro90º )
      I_Contact( #Giro180º )
      I_Contact( #Giro270º )
      Move(in := #V_TOut_MG_90º, out1 => #V_TOut_MG)
   END_RUNG
   // the same network as SCL:
   IF "ON" AND #Giro90º THEN #V_TOut_MG := #V_TOut_MG_90º; END_IF;
   IF "ON" AND #Giro180º THEN #V_TOut_MG := #V_TOut_MG_180º; END_IF;
   IF "ON" AND #Giro270º THEN #V_TOut_MG := #V_TOut_MG_270º; END_IF;
   IF "ON" AND NOT #Giro90º AND NOT #Giro180º AND NOT #Giro270º THEN #V_TOut_MG := #V_TOut_MG_90º; END_IF;
END_REGION

REGION Network 23: ERROR - Timeout Giro (2/4)
   RUNG wire#powerrail
      #TOut_MG(IN := wire#w3, R := wire#w4, PV := #V_TOut_MG, BaseUnidades_ms := "CTE_BaseUnidades_1s", QU =>, QD =>, CVU =>, CVD =>)
   END_RUNG
   RUNG wire#powerrail
      I_Contact( #EstadoZona.Manual_CBx )
      wire#w1
      Contact( #MA_Avance_MG )
      wire#w2
      Contact( #MG_EnMovimiento )
      I_Contact( #Busq_Posicion )
   END_RUNG wire#w3
   RUNG wire#w1
      Contact( #MA_Retroceso_MG )
   END_RUNG wire#w2
   RUNG wire#powerrail
      I_Contact( #MG_EnMovimiento )
   END_RUNG wire#w4
   // the same network as SCL:
   #TOut_MG(IN := NOT #EstadoZona.Manual_CBx AND (#MA_Avance_MG OR #MA_Retroceso_MG) AND #MG_EnMovimiento AND NOT #Busq_Posicion,   // "FB910_CNT_UHS"
            R := NOT #MG_EnMovimiento,
            PV := #V_TOut_MG,
            BaseUnidades_ms := "CTE_BaseUnidades_1s");
END_REGION

REGION Network 24: ERROR - Timeout Giro (3/4)
   // Tiempo máximo de busqueda de posición (mesa en posición desconocida)
   RUNG wire#powerrail
      #TOut_MG_BusPos(IN := wire#w3, R := wire#w4, PV := #V_TOut_MG_BusqPos, BaseUnidades_ms := "CTE_BaseUnidades_1s", QU =>, QD =>, CVU =>, CVD =>)
   END_RUNG
   RUNG wire#powerrail
      I_Contact( #EstadoZona.Manual_CBx )
      wire#w1
      Contact( #MA_Avance_MG )
      wire#w2
      Contact( #MG_EnMovimiento )
      Contact( #Busq_Posicion )
   END_RUNG wire#w3
   RUNG wire#w1
      Contact( #MA_Retroceso_MG )
   END_RUNG wire#w2
   RUNG wire#powerrail
      I_Contact( #MG_EnMovimiento )
   END_RUNG wire#w4
   // the same network as SCL:
   #TOut_MG_BusPos(IN := NOT #EstadoZona.Manual_CBx AND (#MA_Avance_MG OR #MA_Retroceso_MG) AND #MG_EnMovimiento AND #Busq_Posicion,   // "FB910_CNT_UHS"
                   R := NOT #MG_EnMovimiento,
                   PV := #V_TOut_MG_BusqPos,
                   BaseUnidades_ms := "CTE_BaseUnidades_1s");
END_REGION

REGION Network 25: ERROR - Timeout Giro (4/4)
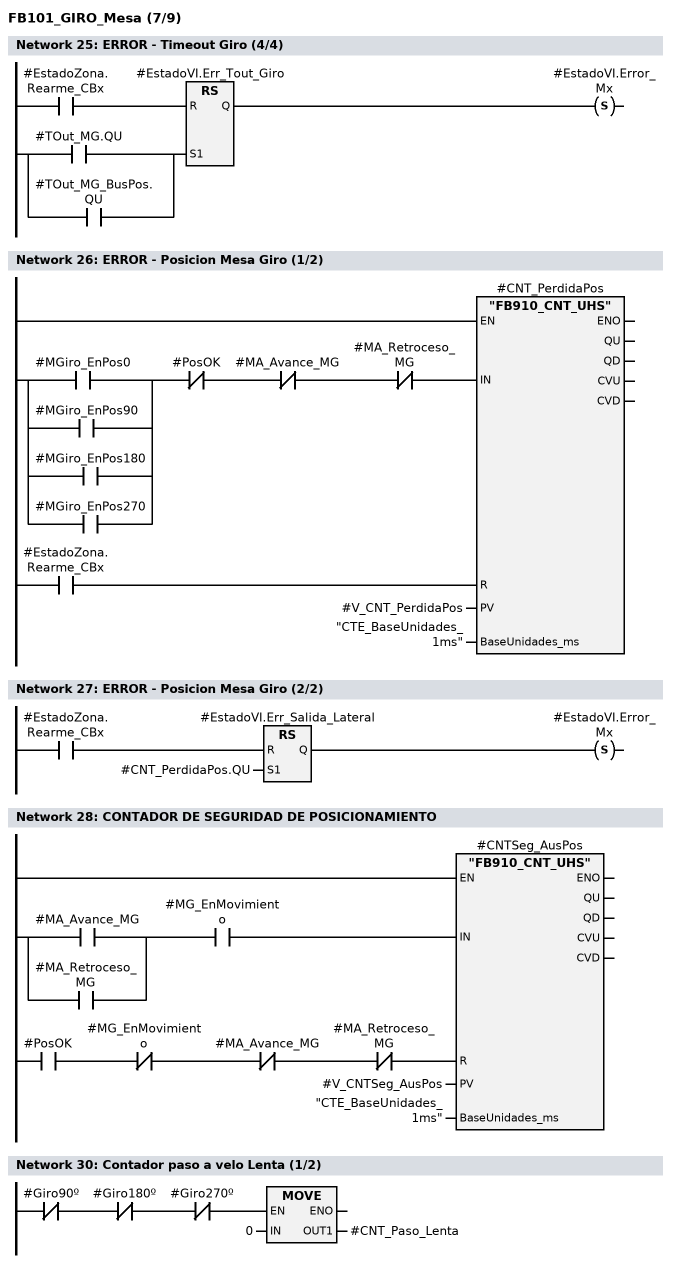
   RUNG wire#powerrail
      Contact( #EstadoZona.Rearme_CBx )
      S_RS(operand := #EstadoVI.Err_Tout_Giro, s1 := wire#w1)
      S_Coil( #EstadoVI.Error_Mx )
   END_RUNG
   RUNG wire#powerrail
      Contact( #TOut_MG.QU )
   END_RUNG wire#w1
   RUNG wire#powerrail
      Contact( #TOut_MG_BusPos.QU )
   END_RUNG wire#w1
   // the same network as SCL:
   IF #EstadoZona.Rearme_CBx THEN
       #EstadoVI.Err_Tout_Giro := FALSE;   // RS flip-flop
   END_IF;
   IF #TOut_MG.QU OR #TOut_MG_BusPos.QU THEN #EstadoVI.Err_Tout_Giro := TRUE; END_IF;
   IF #EstadoVI.Err_Tout_Giro THEN #EstadoVI.Error_Mx := TRUE; END_IF;
END_REGION

REGION Network 26: ERROR - Posicion Mesa Giro (1/2)
   RUNG wire#powerrail
      #CNT_PerdidaPos(IN := wire#w2, R := wire#w3, PV := #V_CNT_PerdidaPos, BaseUnidades_ms := "CTE_BaseUnidades_1ms", QU =>, QD =>, CVU =>, CVD =>)
   END_RUNG
   RUNG wire#powerrail
      Contact( #MGiro_EnPos0 )
      wire#w1
      I_Contact( #PosOK )
      I_Contact( #MA_Avance_MG )
      I_Contact( #MA_Retroceso_MG )
   END_RUNG wire#w2
   RUNG wire#powerrail
      Contact( #MGiro_EnPos90 )
   END_RUNG wire#w1
   RUNG wire#powerrail
      Contact( #MGiro_EnPos180 )
   END_RUNG wire#w1
   RUNG wire#powerrail
      Contact( #MGiro_EnPos270 )
   END_RUNG wire#w1
   RUNG wire#powerrail
      Contact( #EstadoZona.Rearme_CBx )
   END_RUNG wire#w3
   // the same network as SCL:
   #CNT_PerdidaPos(IN := (#MGiro_EnPos0 OR #MGiro_EnPos90 OR #MGiro_EnPos180 OR #MGiro_EnPos270) AND NOT #PosOK AND NOT #MA_Avance_MG AND NOT #MA_Retroceso_MG,   // "FB910_CNT_UHS"
                   R := #EstadoZona.Rearme_CBx,
                   PV := #V_CNT_PerdidaPos,
                   BaseUnidades_ms := "CTE_BaseUnidades_1ms");
END_REGION

REGION Network 27: ERROR - Posicion Mesa Giro (2/2)
   RUNG wire#powerrail
      Contact( #EstadoZona.Rearme_CBx )
      S_RS(operand := #EstadoVI.Err_Salida_Lateral, s1 := #CNT_PerdidaPos.QU)
      S_Coil( #EstadoVI.Error_Mx )
   END_RUNG
   // the same network as SCL:
   IF #EstadoZona.Rearme_CBx THEN
       #EstadoVI.Err_Salida_Lateral := FALSE;   // RS flip-flop
   END_IF;
   IF #CNT_PerdidaPos.QU THEN #EstadoVI.Err_Salida_Lateral := TRUE; END_IF;
   IF #EstadoVI.Err_Salida_Lateral THEN #EstadoVI.Error_Mx := TRUE; END_IF;
END_REGION

REGION Network 28: CONTADOR DE SEGURIDAD DE POSICIONAMIENTO
   RUNG wire#powerrail
      #CNTSeg_AusPos(IN := wire#w2, R := wire#w3, PV := #V_CNTSeg_AusPos, BaseUnidades_ms := "CTE_BaseUnidades_1ms", QU =>, QD =>, CVU =>, CVD =>)
   END_RUNG
   RUNG wire#powerrail
      Contact( #MA_Avance_MG )
      wire#w1
      Contact( #MG_EnMovimiento )
   END_RUNG wire#w2
   RUNG wire#powerrail
      Contact( #MA_Retroceso_MG )
   END_RUNG wire#w1
   RUNG wire#powerrail
      Contact( #PosOK )
      I_Contact( #MG_EnMovimiento )
      I_Contact( #MA_Avance_MG )
      I_Contact( #MA_Retroceso_MG )
   END_RUNG wire#w3
   // the same network as SCL:
   #CNTSeg_AusPos(IN := (#MA_Avance_MG OR #MA_Retroceso_MG) AND #MG_EnMovimiento,   // "FB910_CNT_UHS"
                  R := #PosOK AND NOT #MG_EnMovimiento AND NOT #MA_Avance_MG AND NOT #MA_Retroceso_MG,
                  PV := #V_CNTSeg_AusPos,
                  BaseUnidades_ms := "CTE_BaseUnidades_1ms");
END_REGION

REGION Network 29: CONTADOR DE VELOCIDAD LENTA
END_REGION

REGION Network 30: Contador paso a velo Lenta (1/2)
   RUNG wire#powerrail
      I_Contact( #Giro90º )
      I_Contact( #Giro180º )
      I_Contact( #Giro270º )
      { S7_GenerateENO := "TRUE" } Move(in := 0, out1 => #CNT_Paso_Lenta)
   END_RUNG
   // the same network as SCL:
   IF NOT #Giro90º AND NOT #Giro180º AND NOT #Giro270º THEN #CNT_Paso_Lenta := 0; END_IF;
END_REGION

REGION Network 31: Contador paso a velo Lenta (2/2)
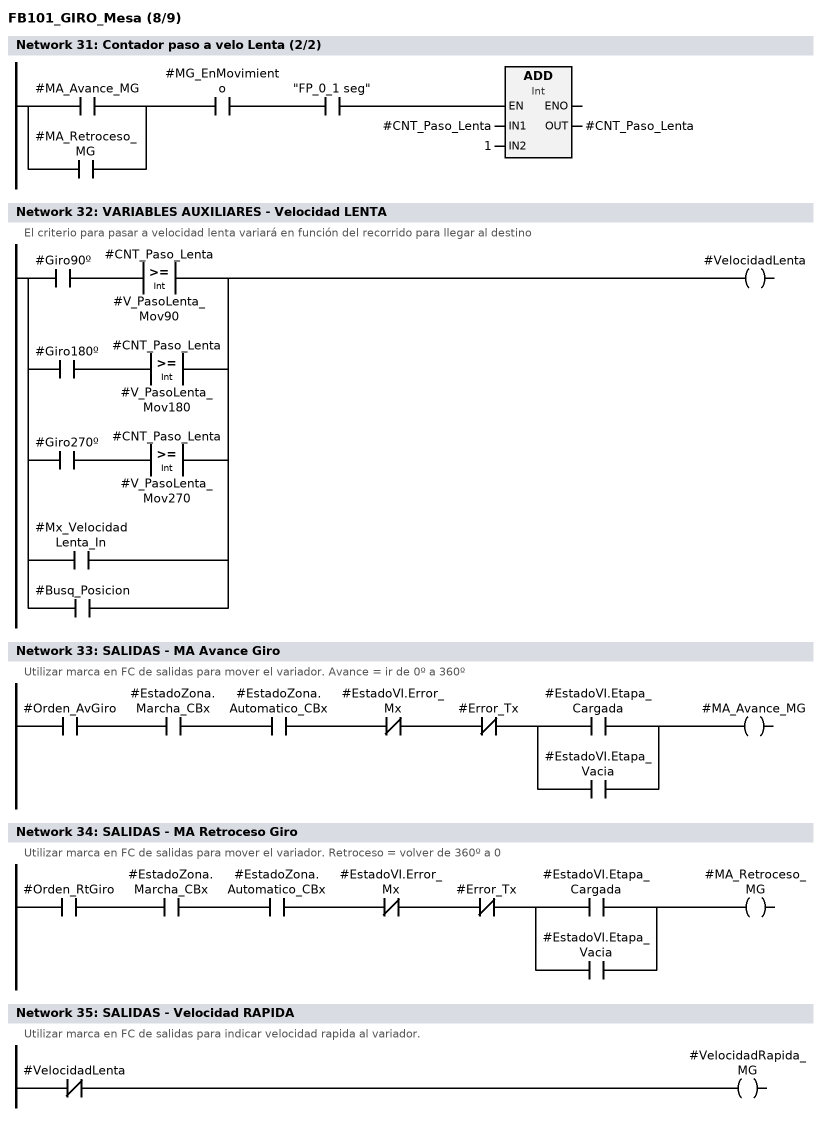
   RUNG wire#powerrail
      Contact( #MA_Avance_MG )
      wire#w1
      Contact( #MG_EnMovimiento )
      Contact( "FP_0_1 seg" )
      { S7_Templates := "SrcType := Int"; S7_GenerateENO := "TRUE" } Add(in1 := #CNT_Paso_Lenta, in2 := 1, out => #CNT_Paso_Lenta)
   END_RUNG
   RUNG wire#powerrail
      Contact( #MA_Retroceso_MG )
   END_RUNG wire#w1
   // the same network as SCL:
   IF (#MA_Avance_MG OR #MA_Retroceso_MG) AND #MG_EnMovimiento AND "FP_0_1 seg" THEN
       #CNT_Paso_Lenta := #CNT_Paso_Lenta + 1;
   END_IF;
END_REGION

REGION Network 32: VARIABLES AUXILIARES - Velocidad LENTA
   // El criterio para pasar a velocidad lenta variará en función del recorrido para llegar al destino
   RUNG wire#powerrail
      Contact( #Giro90º )
      { S7_Templates := "SrcType := Int" } GE_Contact(in1 := #CNT_Paso_Lenta, in2 := #V_PasoLenta_Mov90)
      wire#w1
      Coil( #VelocidadLenta )
   END_RUNG
   RUNG wire#powerrail
      Contact( #Giro180º )
      { S7_Templates := "SrcType := Int" } GE_Contact(in1 := #CNT_Paso_Lenta, in2 := #V_PasoLenta_Mov180)
   END_RUNG wire#w1
   RUNG wire#powerrail
      Contact( #Giro270º )
      { S7_Templates := "SrcType := Int" } GE_Contact(in1 := #CNT_Paso_Lenta, in2 := #V_PasoLenta_Mov270)
   END_RUNG wire#w1
   RUNG wire#powerrail
      Contact( #Mx_VelocidadLenta_In )
   END_RUNG wire#w1
   RUNG wire#powerrail
      Contact( #Busq_Posicion )
   END_RUNG wire#w1
   // the same network as SCL:
   #VelocidadLenta := (#Giro90º AND (#CNT_Paso_Lenta >= #V_PasoLenta_Mov90)) OR (#Giro180º AND (#CNT_Paso_Lenta >= #V_PasoLenta_Mov180)) OR (#Giro270º AND (#CNT_Paso_Lenta >= #V_PasoLenta_Mov270)) OR #Mx_VelocidadLenta_In OR #Busq_Posicion;
END_REGION

REGION Network 33: SALIDAS - MA Avance Giro
   // Utilizar marca en FC de salidas para mover el variador. Avance = ir de 0º a 360º
   RUNG wire#powerrail
      Contact( #Orden_AvGiro )
      Contact( #EstadoZona.Marcha_CBx )
      Contact( #EstadoZona.Automatico_CBx )
      I_Contact( #EstadoVI.Error_Mx )
      I_Contact( #Error_Tx )
      wire#w1
      Contact( #EstadoVI.Etapa_Cargada )
      wire#w2
      Coil( #MA_Avance_MG )
   END_RUNG
   RUNG wire#w1
      Contact( #EstadoVI.Etapa_Vacia )
   END_RUNG wire#w2
   // the same network as SCL:
   #MA_Avance_MG := #Orden_AvGiro AND #EstadoZona.Marcha_CBx AND #EstadoZona.Automatico_CBx AND NOT #EstadoVI.Error_Mx AND NOT #Error_Tx AND (#EstadoVI.Etapa_Cargada OR #EstadoVI.Etapa_Vacia);
END_REGION

REGION Network 34: SALIDAS - MA Retroceso Giro
   // Utilizar marca en FC de salidas para mover el variador. Retroceso = volver de 360º a 0
   RUNG wire#powerrail
      Contact( #Orden_RtGiro )
      Contact( #EstadoZona.Marcha_CBx )
      Contact( #EstadoZona.Automatico_CBx )
      I_Contact( #EstadoVI.Error_Mx )
      I_Contact( #Error_Tx )
      wire#w1
      Contact( #EstadoVI.Etapa_Cargada )
      wire#w2
      Coil( #MA_Retroceso_MG )
   END_RUNG
   RUNG wire#w1
      Contact( #EstadoVI.Etapa_Vacia )
   END_RUNG wire#w2
   // the same network as SCL:
   #MA_Retroceso_MG := #Orden_RtGiro AND #EstadoZona.Marcha_CBx AND #EstadoZona.Automatico_CBx AND NOT #EstadoVI.Error_Mx AND NOT #Error_Tx AND (#EstadoVI.Etapa_Cargada OR #EstadoVI.Etapa_Vacia);
END_REGION

REGION Network 35: SALIDAS - Velocidad RAPIDA
   // Utilizar marca en FC de salidas para indicar velocidad rapida al variador.
   RUNG wire#powerrail
      I_Contact( #VelocidadLenta )
      Coil( #VelocidadRapida_MG )
   END_RUNG
   // the same network as SCL:
   #VelocidadRapida_MG := NOT #VelocidadLenta;
END_REGION

REGION Network 36: ENTRADAS DE LA MESA
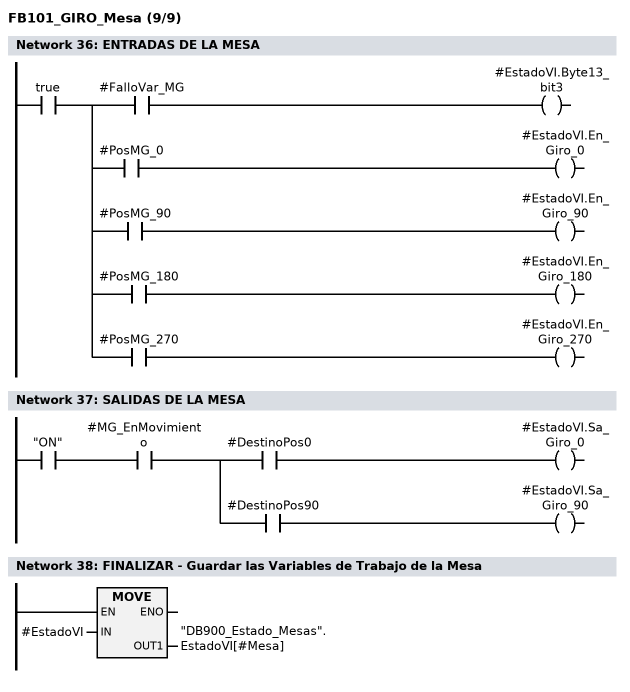
   RUNG wire#powerrail
      Contact( true )
      wire#w1
      Contact( #FalloVar_MG )
      Coil( #EstadoVI.Byte13_bit3 )
   END_RUNG
   RUNG wire#w1
      Contact( #PosMG_0 )
      Coil( #EstadoVI.En_Giro_0 )
   END_RUNG
   RUNG wire#w1
      Contact( #PosMG_90 )
      Coil( #EstadoVI.En_Giro_90 )
   END_RUNG
   RUNG wire#w1
      Contact( #PosMG_180 )
      Coil( #EstadoVI.En_Giro_180 )
   END_RUNG
   RUNG wire#w1
      Contact( #PosMG_270 )
      Coil( #EstadoVI.En_Giro_270 )
   END_RUNG
   // the same network as SCL:
   #EstadoVI.Byte13_bit3 := true AND #FalloVar_MG;
   #EstadoVI.En_Giro_0 := true AND #PosMG_0;
   #EstadoVI.En_Giro_90 := true AND #PosMG_90;
   #EstadoVI.En_Giro_180 := true AND #PosMG_180;
   #EstadoVI.En_Giro_270 := true AND #PosMG_270;
END_REGION

REGION Network 37: SALIDAS DE LA MESA
   RUNG wire#powerrail
      Contact( "ON" )
      Contact( #MG_EnMovimiento )
      wire#w1
      Contact( #DestinoPos0 )
      Coil( #EstadoVI.Sa_Giro_0 )
   END_RUNG
   RUNG wire#w1
      Contact( #DestinoPos90 )
      Coil( #EstadoVI.Sa_Giro_90 )
   END_RUNG
   // the same network as SCL:
   #_w1 := "ON" AND #MG_EnMovimiento;
   #EstadoVI.Sa_Giro_0 := #_w1 AND #DestinoPos0;
   #EstadoVI.Sa_Giro_90 := #_w1 AND #DestinoPos90;
END_REGION

REGION Network 38: FINALIZAR - Guardar las Variables de Trabajo de la Mesa
   RUNG wire#powerrail
      Move(in := #EstadoVI, out1 => "DB900_Estado_Mesas".EstadoVI[#Mesa])
   END_RUNG
   // the same network as SCL:
   "DB900_Estado_Mesas".EstadoVI[#Mesa] := #EstadoVI;
END_REGION
END_FUNCTION_BLOCK
